PROGRAM PackML_U01
VAR
	fbRobotCell			: FB_Robot_U01;
	fbInfeed 			: FB_Infeed_U01_SU01;
	fbDelta				: FB_Delta_U01_SU02;
	fbDischarge			: FB_Discharge_U01_SU03;
	stPMLSubUnitInfo	: ARRAY [1..4] OF ST_PMLSubUnitInfo;	//Informations about the Subunits
END_VAR

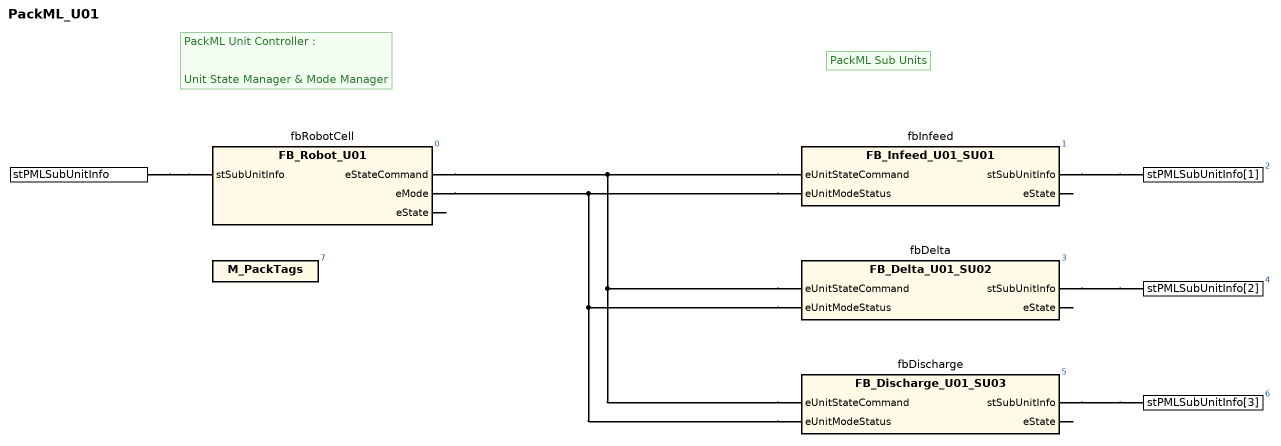
// PackML Unit Controller :
//
// Unit State Manager & Mode Manager
fbRobotCell(stSubUnitInfo := stPMLSubUnitInfo); // FB_Robot_U01
// PackML Sub Units
fbInfeed(eUnitStateCommand := fbRobotCell.eStateCommand, eUnitModeStatus := fbRobotCell.eMode); // FB_Infeed_U01_SU01
stPMLSubUnitInfo[1] := fbInfeed.stSubUnitInfo;
fbDelta(eUnitStateCommand := fbRobotCell.eStateCommand, eUnitModeStatus := fbRobotCell.eMode); // FB_Delta_U01_SU02
stPMLSubUnitInfo[2] := fbDelta.stSubUnitInfo;
fbDischarge(eUnitStateCommand := fbRobotCell.eStateCommand, eUnitModeStatus := fbRobotCell.eMode); // FB_Discharge_U01_SU03
stPMLSubUnitInfo[3] := fbDischarge.stSubUnitInfo;
M_PackTags();

METHOD M_PackTags
VAR_INPUT
END_VAR


// Commands to Unit 01 from the Line Controller
fbRobotCell.P_PackTags.Command := GVL.UnitPackTags[1].Command;

// Status & Admin Data of Unit 01 to the Line Controller
GVL.UnitPackTags[1].Status	:= fbRobotCell.P_PackTags.Status;
GVL.UnitPackTags[1].Admin	:= fbRobotCell.P_PackTags.Admin;
END_METHOD

END_PROGRAM

(* stored: Version 1.1.0.1, ProductVersion 3.1.4024.11
   POU PackML_U01: Id {62ad58c9-195a-4e27-9c10-112e801e44a4}, SpecialFunc None
   Method M_PackTags: Id {d93973e9-cff9-4ba5-807f-9467ca062944} *)
